(*
A list implementation for managing `I_Arg`.  
*)
INTERFACE I_MutArgList EXTENDS I_ArgList

(*
Adds, updates, or removes an argument in the list at the specified index.  
Return:
- `Ok` - Upon successfully adding, modifying, or removing an entry.
- `None` - When replacing a null entry with another null entry.
- `Err.Ovf` - When attempting to modify an entry at an out-of-bounds index.
*)
METHOD Append : Result
VAR_INPUT
	iArg		: I_Arg;
	nIndex		: UDINT;
END_VAR
END_METHOD

END_INTERFACE

(* stored: Version 1.1.0.1
   Itf I_MutArgList: Id {a13a3abf-b20e-494a-a089-922a6c403ef2}
   Method Append: Id {9cd928ff-dfb7-497d-a0a3-0685d1fb0111} *)
